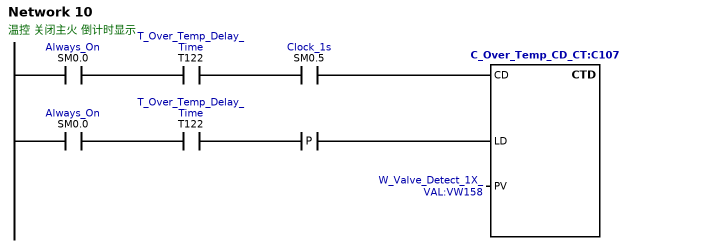
[picture p24: SBR4 networks 10-10]
Network 10
// 温控 关闭主火 倒计时显示
LD     Always_On:SM0.0
A      T_Over_Temp_Delay_Time:T122
A      Clock_1s:SM0.5
LD     Always_On:SM0.0
A      T_Over_Temp_Delay_Time:T122
EU
CTD    C_Over_Temp_CD_CT:C107, W_Valve_Detect_1X_VAL:VW158
END_SUBROUTINE_BLOCK

SUBROUTINE_BLOCK 阶段升温:SBR5
TITLE=
BEGIN
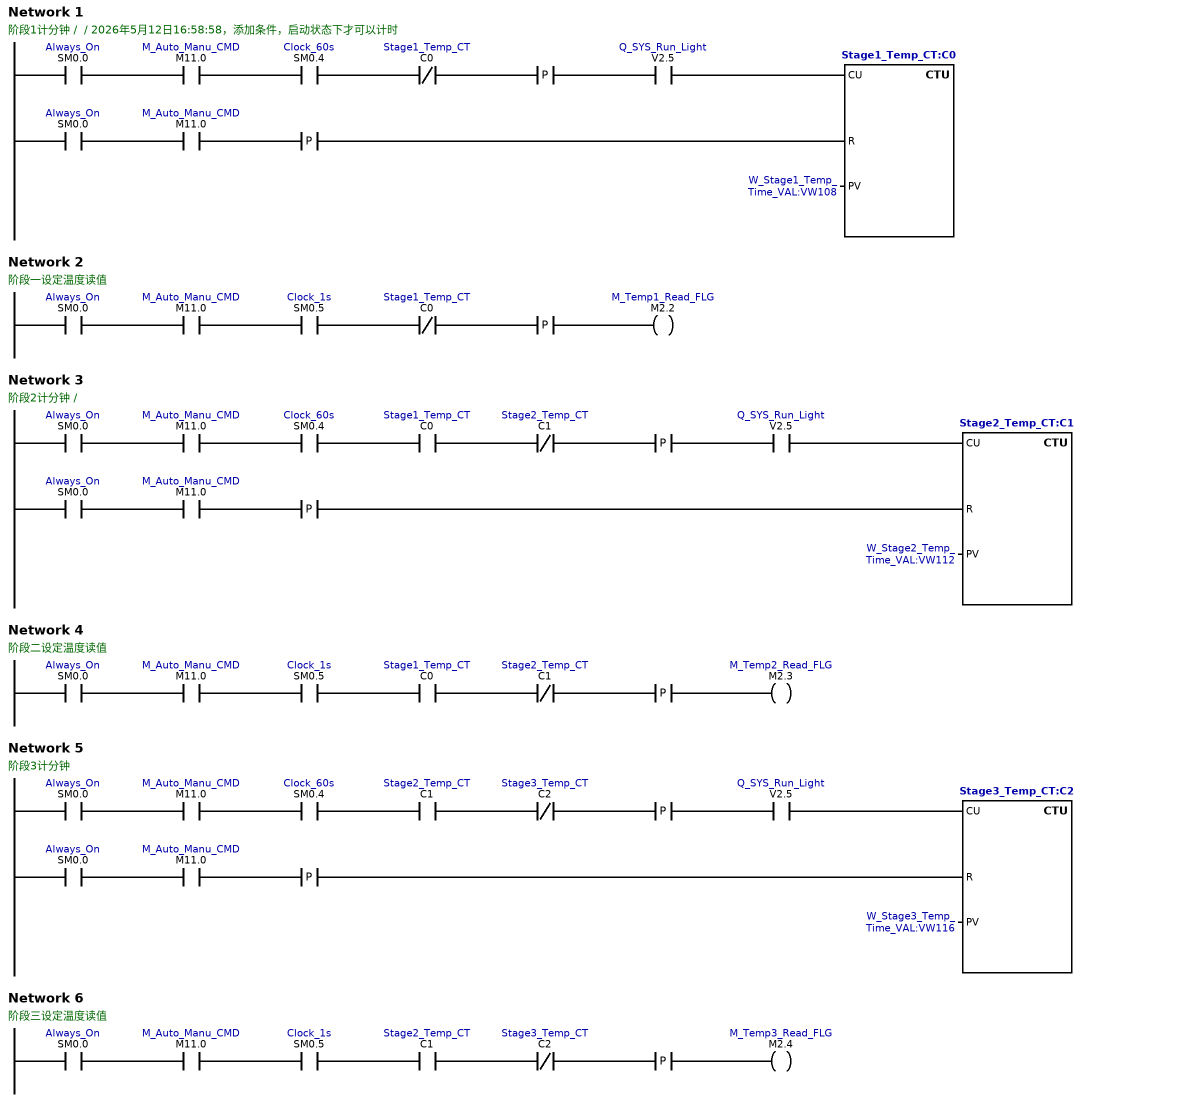
Network 1
// 阶段1计分钟
// 
// 2026年5月12日16:58:58，添加条件，启动状态下才可以计时
LD     Always_On:SM0.0
A      M_Auto_Manu_CMD:M11.0
A      Clock_60s:SM0.4
AN     Stage1_Temp_CT:C0
EU
A      Q_SYS_Run_Light:V2.5
LD     Always_On:SM0.0
A      M_Auto_Manu_CMD:M11.0
EU
CTU    Stage1_Temp_CT:C0, W_Stage1_Temp_Time_VAL:VW108
Network 2
// 阶段一设定温度读值
LD     Always_On:SM0.0
A      M_Auto_Manu_CMD:M11.0
A      Clock_1s:SM0.5
AN     Stage1_Temp_CT:C0
EU
=      M_Temp1_Read_FLG:M2.2
Network 3
// 阶段2计分钟
// 
LD     Always_On:SM0.0
A      M_Auto_Manu_CMD:M11.0
A      Clock_60s:SM0.4
A      Stage1_Temp_CT:C0
AN     Stage2_Temp_CT:C1
EU
A      Q_SYS_Run_Light:V2.5
LD     Always_On:SM0.0
A      M_Auto_Manu_CMD:M11.0
EU
CTU    Stage2_Temp_CT:C1, W_Stage2_Temp_Time_VAL:VW112
Network 4
// 阶段二设定温度读值
LD     Always_On:SM0.0
A      M_Auto_Manu_CMD:M11.0
A      Clock_1s:SM0.5
A      Stage1_Temp_CT:C0
AN     Stage2_Temp_CT:C1
EU
=      M_Temp2_Read_FLG:M2.3
Network 5
// 阶段3计分钟
LD     Always_On:SM0.0
A      M_Auto_Manu_CMD:M11.0
A      Clock_60s:SM0.4
A      Stage2_Temp_CT:C1
AN     Stage3_Temp_CT:C2
EU
A      Q_SYS_Run_Light:V2.5
LD     Always_On:SM0.0
A      M_Auto_Manu_CMD:M11.0
EU
CTU    Stage3_Temp_CT:C2, W_Stage3_Temp_Time_VAL:VW116
Network 6
// 阶段三设定温度读值
LD     Always_On:SM0.0
A      M_Auto_Manu_CMD:M11.0
A      Clock_1s:SM0.5
A      Stage2_Temp_CT:C1
AN     Stage3_Temp_CT:C2
EU
=      M_Temp3_Read_FLG:M2.4
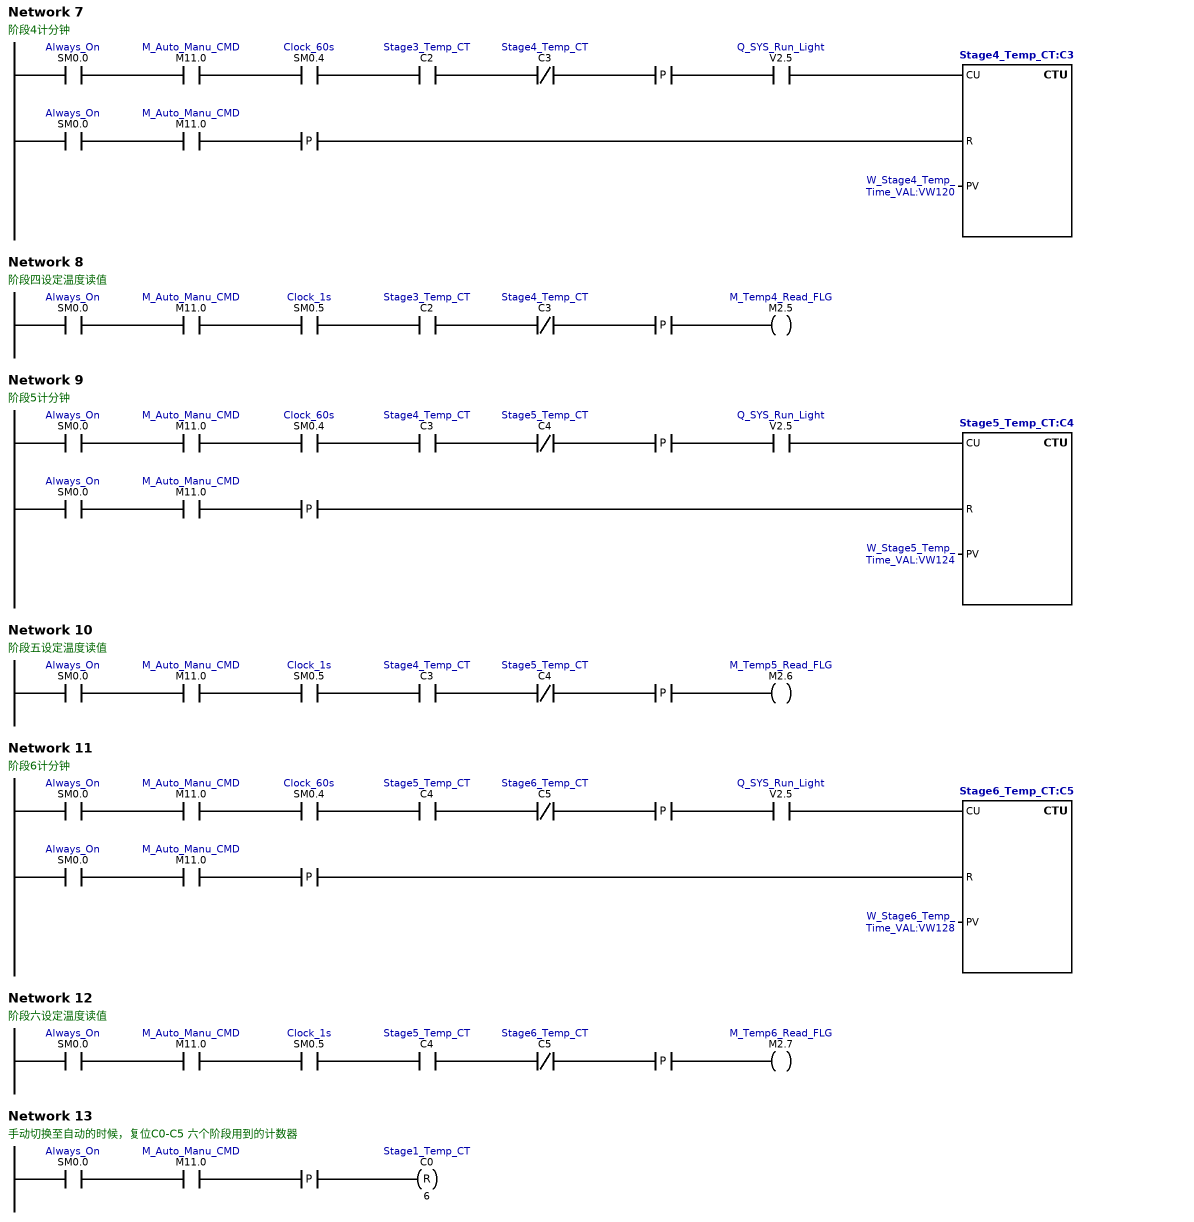
Network 7
// 阶段4计分钟
LD     Always_On:SM0.0
A      M_Auto_Manu_CMD:M11.0
A      Clock_60s:SM0.4
A      Stage3_Temp_CT:C2
AN     Stage4_Temp_CT:C3
EU
A      Q_SYS_Run_Light:V2.5
LD     Always_On:SM0.0
A      M_Auto_Manu_CMD:M11.0
EU
CTU    Stage4_Temp_CT:C3, W_Stage4_Temp_Time_VAL:VW120
Network 8
// 阶段四设定温度读值
LD     Always_On:SM0.0
A      M_Auto_Manu_CMD:M11.0
A      Clock_1s:SM0.5
A      Stage3_Temp_CT:C2
AN     Stage4_Temp_CT:C3
EU
=      M_Temp4_Read_FLG:M2.5
Network 9
// 阶段5计分钟
LD     Always_On:SM0.0
A      M_Auto_Manu_CMD:M11.0
A      Clock_60s:SM0.4
A      Stage4_Temp_CT:C3
AN     Stage5_Temp_CT:C4
EU
A      Q_SYS_Run_Light:V2.5
LD     Always_On:SM0.0
A      M_Auto_Manu_CMD:M11.0
EU
CTU    Stage5_Temp_CT:C4, W_Stage5_Temp_Time_VAL:VW124
Network 10
// 阶段五设定温度读值
LD     Always_On:SM0.0
A      M_Auto_Manu_CMD:M11.0
A      Clock_1s:SM0.5
A      Stage4_Temp_CT:C3
AN     Stage5_Temp_CT:C4
EU
=      M_Temp5_Read_FLG:M2.6
Network 11
// 阶段6计分钟
LD     Always_On:SM0.0
A      M_Auto_Manu_CMD:M11.0
A      Clock_60s:SM0.4
A      Stage5_Temp_CT:C4
AN     Stage6_Temp_CT:C5
EU
A      Q_SYS_Run_Light:V2.5
LD     Always_On:SM0.0
A      M_Auto_Manu_CMD:M11.0
EU
CTU    Stage6_Temp_CT:C5, W_Stage6_Temp_Time_VAL:VW128
Network 12
// 阶段六设定温度读值
LD     Always_On:SM0.0
A      M_Auto_Manu_CMD:M11.0
A      Clock_1s:SM0.5
A      Stage5_Temp_CT:C4
AN     Stage6_Temp_CT:C5
EU
=      M_Temp6_Read_FLG:M2.7
Network 13
// 手动切换至自动的时候，复位C0-C5 六个阶段用到的计数器
LD     Always_On:SM0.0
A      M_Auto_Manu_CMD:M11.0
EU
R      Stage1_Temp_CT:C0, 6
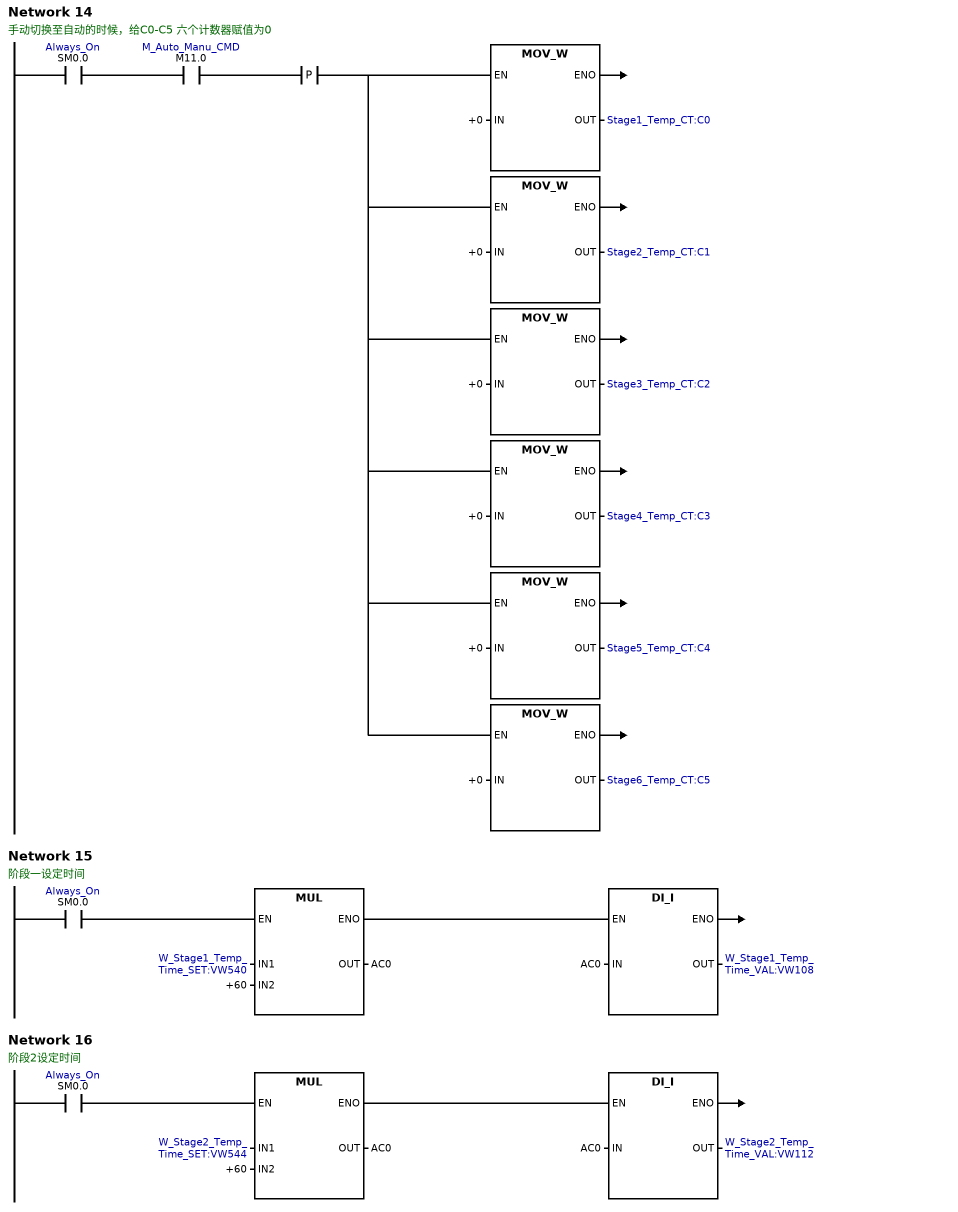
Network 14
// 手动切换至自动的时候，给C0-C5 六个计数器赋值为0
LD     Always_On:SM0.0
A      M_Auto_Manu_CMD:M11.0
EU
MOVW   +0, Stage1_Temp_CT:C0
MOVW   +0, Stage2_Temp_CT:C1
MOVW   +0, Stage3_Temp_CT:C2
MOVW   +0, Stage4_Temp_CT:C3
MOVW   +0, Stage5_Temp_CT:C4
MOVW   +0, Stage6_Temp_CT:C5
Network 15
// 阶段一设定时间
LD     Always_On:SM0.0
MOVW   W_Stage1_Temp_Time_SET:VW540, AC0
AENO
MUL    +60, AC0
AENO
DTI    AC0, W_Stage1_Temp_Time_VAL:VW108
Network 16
// 阶段2设定时间
LD     Always_On:SM0.0
MOVW   W_Stage2_Temp_Time_SET:VW544, AC0
AENO
MUL    +60, AC0
AENO
DTI    AC0, W_Stage2_Temp_Time_VAL:VW112
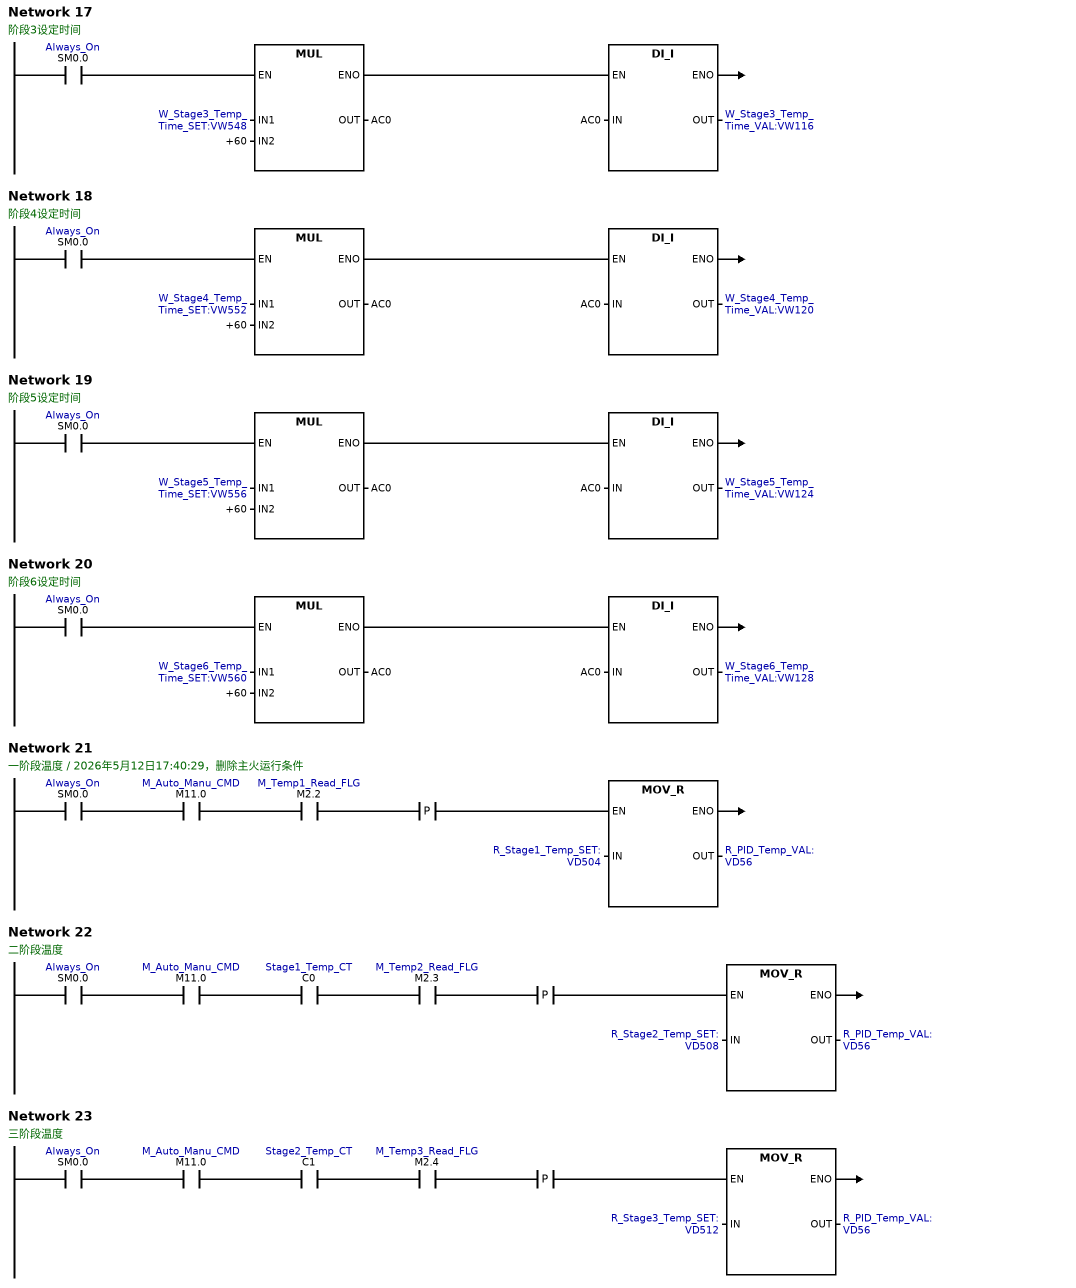
Network 17
// 阶段3设定时间
LD     Always_On:SM0.0
MOVW   W_Stage3_Temp_Time_SET:VW548, AC0
AENO
MUL    +60, AC0
AENO
DTI    AC0, W_Stage3_Temp_Time_VAL:VW116
Network 18
// 阶段4设定时间
LD     Always_On:SM0.0
MOVW   W_Stage4_Temp_Time_SET:VW552, AC0
AENO
MUL    +60, AC0
AENO
DTI    AC0, W_Stage4_Temp_Time_VAL:VW120
Network 19
// 阶段5设定时间
LD     Always_On:SM0.0
MOVW   W_Stage5_Temp_Time_SET:VW556, AC0
AENO
MUL    +60, AC0
AENO
DTI    AC0, W_Stage5_Temp_Time_VAL:VW124
Network 20
// 阶段6设定时间
LD     Always_On:SM0.0
MOVW   W_Stage6_Temp_Time_SET:VW560, AC0
AENO
MUL    +60, AC0
AENO
DTI    AC0, W_Stage6_Temp_Time_VAL:VW128
Network 21
// 一阶段温度
// 2026年5月12日17:40:29，删除主火运行条件
LD     Always_On:SM0.0
A      M_Auto_Manu_CMD:M11.0
A      M_Temp1_Read_FLG:M2.2
EU
MOVR   R_Stage1_Temp_SET:VD504, R_PID_Temp_VAL:VD56
Network 22
// 二阶段温度
LD     Always_On:SM0.0
A      M_Auto_Manu_CMD:M11.0
A      Stage1_Temp_CT:C0
A      M_Temp2_Read_FLG:M2.3
EU
MOVR   R_Stage2_Temp_SET:VD508, R_PID_Temp_VAL:VD56
Network 23
// 三阶段温度
LD     Always_On:SM0.0
A      M_Auto_Manu_CMD:M11.0
A      Stage2_Temp_CT:C1
A      M_Temp3_Read_FLG:M2.4
EU
MOVR   R_Stage3_Temp_SET:VD512, R_PID_Temp_VAL:VD56
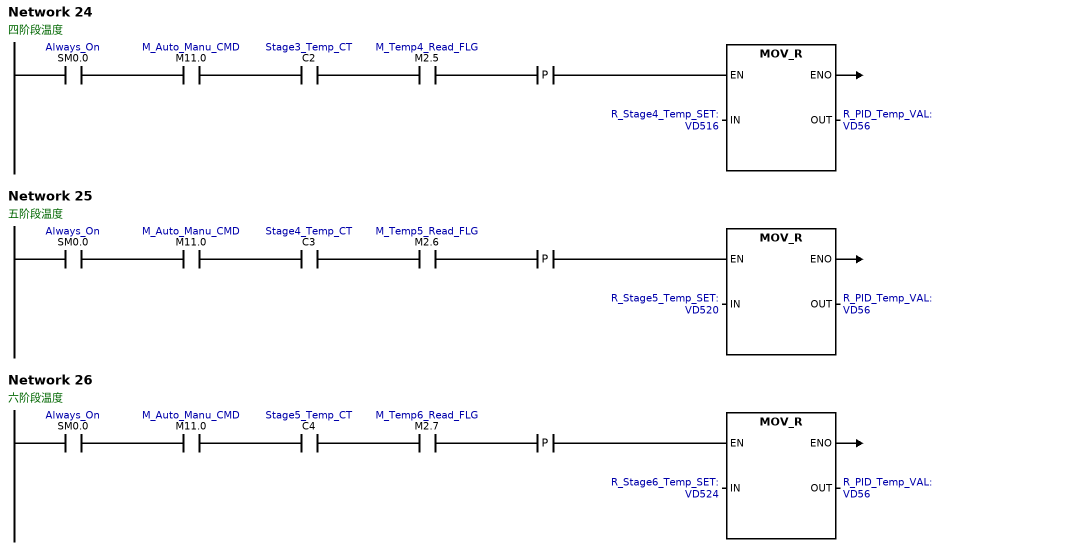
Network 24
// 四阶段温度
LD     Always_On:SM0.0
A      M_Auto_Manu_CMD:M11.0
A      Stage3_Temp_CT:C2
A      M_Temp4_Read_FLG:M2.5
EU
MOVR   R_Stage4_Temp_SET:VD516, R_PID_Temp_VAL:VD56
Network 25
// 五阶段温度
LD     Always_On:SM0.0
A      M_Auto_Manu_CMD:M11.0
A      Stage4_Temp_CT:C3
A      M_Temp5_Read_FLG:M2.6
EU
MOVR   R_Stage5_Temp_SET:VD520, R_PID_Temp_VAL:VD56
Network 26
// 六阶段温度
LD     Always_On:SM0.0
A      M_Auto_Manu_CMD:M11.0
A      Stage5_Temp_CT:C4
A      M_Temp6_Read_FLG:M2.7
EU
MOVR   R_Stage6_Temp_SET:VD524, R_PID_Temp_VAL:VD56
END_SUBROUTINE_BLOCK

SUBROUTINE_BLOCK 开度档位:SBR6
TITLE=开度档位子程序
// 功能：
// 1、处理每档对应的燃气调节阀开度多少，空气调节阀开度多少。
// 2、手动模式，升档、降档控制
// 3、自动模式，PID输出转换成档位处理
// 
BEGIN
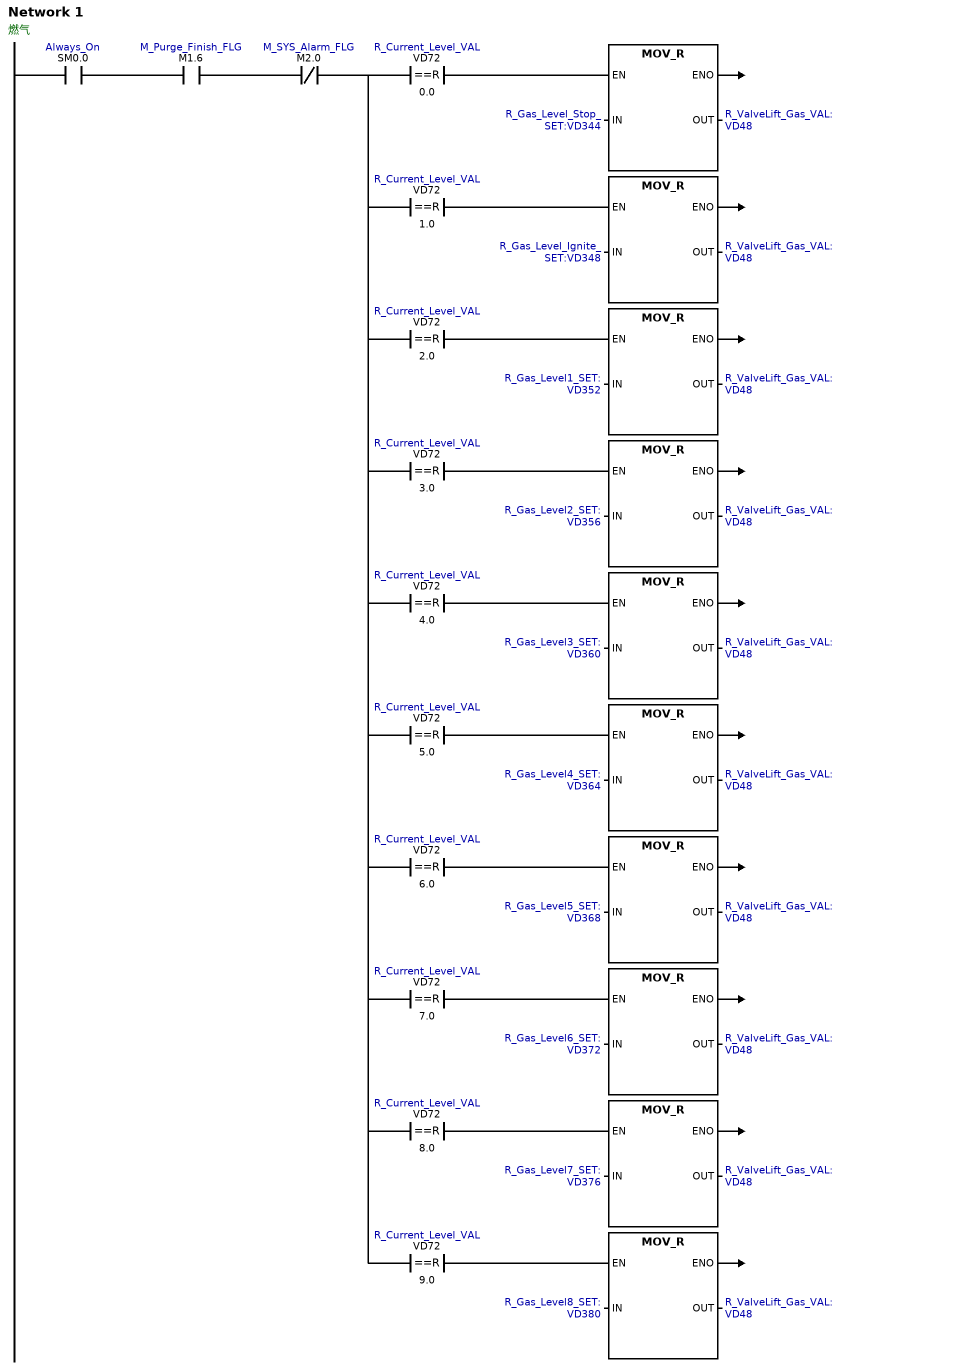
Network 1
// 燃气
LD     Always_On:SM0.0
A      M_Purge_Finish_FLG:M1.6
AN     M_SYS_Alarm_FLG:M2.0
LPS
AR=    R_Current_Level_VAL:VD72, 0.0
MOVR   R_Gas_Level_Stop_SET:VD344, R_ValveLift_Gas_VAL:VD48
LRD
AR=    R_Current_Level_VAL:VD72, 1.0
MOVR   R_Gas_Level_Ignite_SET:VD348, R_ValveLift_Gas_VAL:VD48
LRD
AR=    R_Current_Level_VAL:VD72, 2.0
MOVR   R_Gas_Level1_SET:VD352, R_ValveLift_Gas_VAL:VD48
LRD
AR=    R_Current_Level_VAL:VD72, 3.0
MOVR   R_Gas_Level2_SET:VD356, R_ValveLift_Gas_VAL:VD48
LRD
AR=    R_Current_Level_VAL:VD72, 4.0
MOVR   R_Gas_Level3_SET:VD360, R_ValveLift_Gas_VAL:VD48
LRD
AR=    R_Current_Level_VAL:VD72, 5.0
MOVR   R_Gas_Level4_SET:VD364, R_ValveLift_Gas_VAL:VD48
LRD
AR=    R_Current_Level_VAL:VD72, 6.0
MOVR   R_Gas_Level5_SET:VD368, R_ValveLift_Gas_VAL:VD48
LRD
AR=    R_Current_Level_VAL:VD72, 7.0
MOVR   R_Gas_Level6_SET:VD372, R_ValveLift_Gas_VAL:VD48
LRD
AR=    R_Current_Level_VAL:VD72, 8.0
MOVR   R_Gas_Level7_SET:VD376, R_ValveLift_Gas_VAL:VD48
LPP
AR=    R_Current_Level_VAL:VD72, 9.0
MOVR   R_Gas_Level8_SET:VD380, R_ValveLift_Gas_VAL:VD48
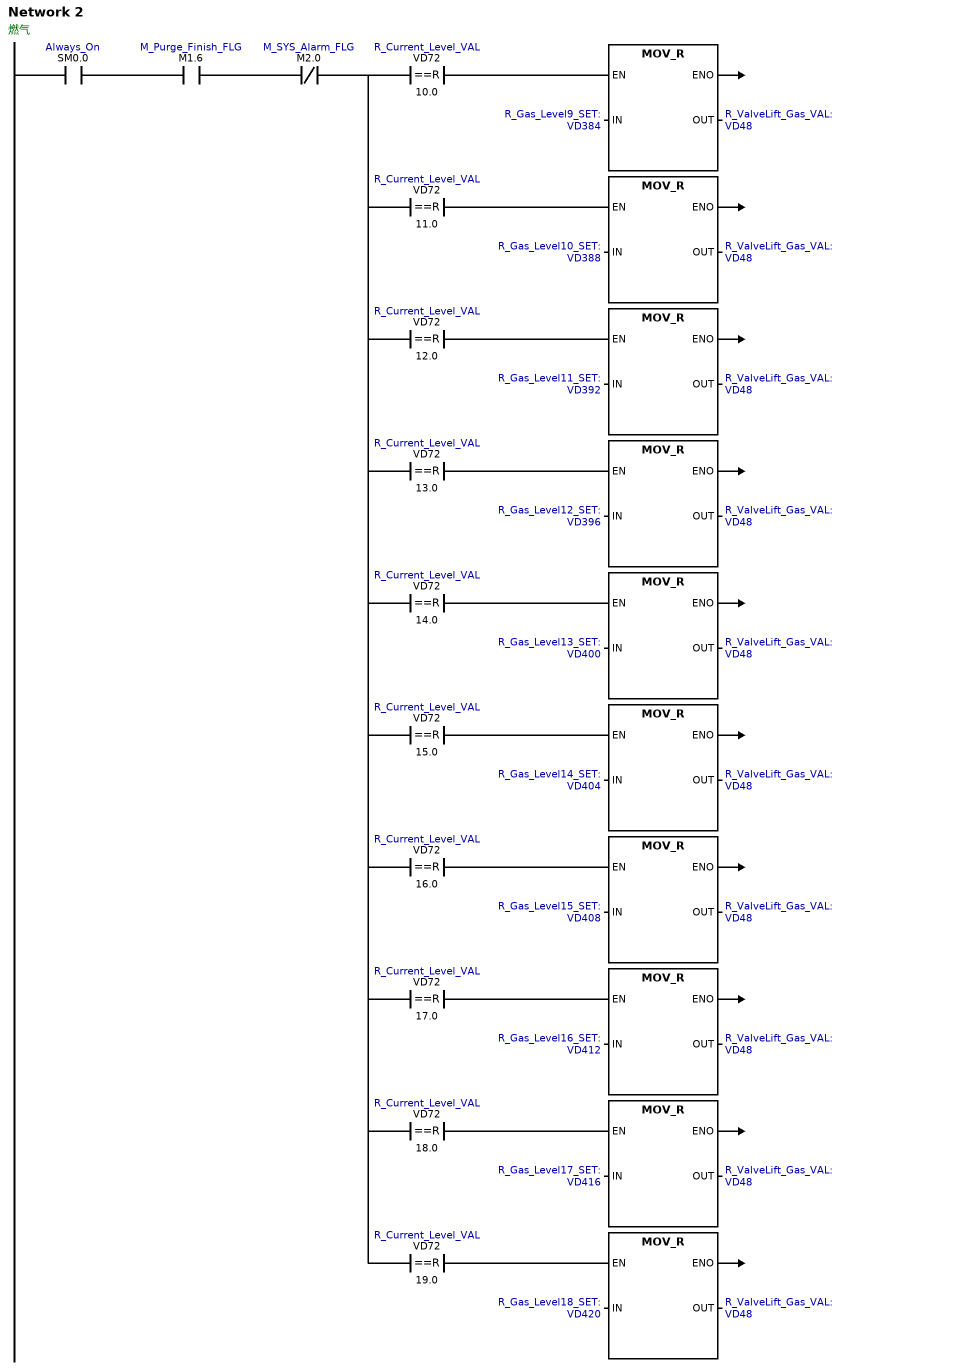
Network 2
// 燃气
LD     Always_On:SM0.0
A      M_Purge_Finish_FLG:M1.6
AN     M_SYS_Alarm_FLG:M2.0
LPS
AR=    R_Current_Level_VAL:VD72, 10.0
MOVR   R_Gas_Level9_SET:VD384, R_ValveLift_Gas_VAL:VD48
LRD
AR=    R_Current_Level_VAL:VD72, 11.0
MOVR   R_Gas_Level10_SET:VD388, R_ValveLift_Gas_VAL:VD48
LRD
AR=    R_Current_Level_VAL:VD72, 12.0
MOVR   R_Gas_Level11_SET:VD392, R_ValveLift_Gas_VAL:VD48
LRD
AR=    R_Current_Level_VAL:VD72, 13.0
MOVR   R_Gas_Level12_SET:VD396, R_ValveLift_Gas_VAL:VD48
LRD
AR=    R_Current_Level_VAL:VD72, 14.0
MOVR   R_Gas_Level13_SET:VD400, R_ValveLift_Gas_VAL:VD48
LRD
AR=    R_Current_Level_VAL:VD72, 15.0
MOVR   R_Gas_Level14_SET:VD404, R_ValveLift_Gas_VAL:VD48
LRD
AR=    R_Current_Level_VAL:VD72, 16.0
MOVR   R_Gas_Level15_SET:VD408, R_ValveLift_Gas_VAL:VD48
LRD
AR=    R_Current_Level_VAL:VD72, 17.0
MOVR   R_Gas_Level16_SET:VD412, R_ValveLift_Gas_VAL:VD48
LRD
AR=    R_Current_Level_VAL:VD72, 18.0
MOVR   R_Gas_Level17_SET:VD416, R_ValveLift_Gas_VAL:VD48
LPP
AR=    R_Current_Level_VAL:VD72, 19.0
MOVR   R_Gas_Level18_SET:VD420, R_ValveLift_Gas_VAL:VD48
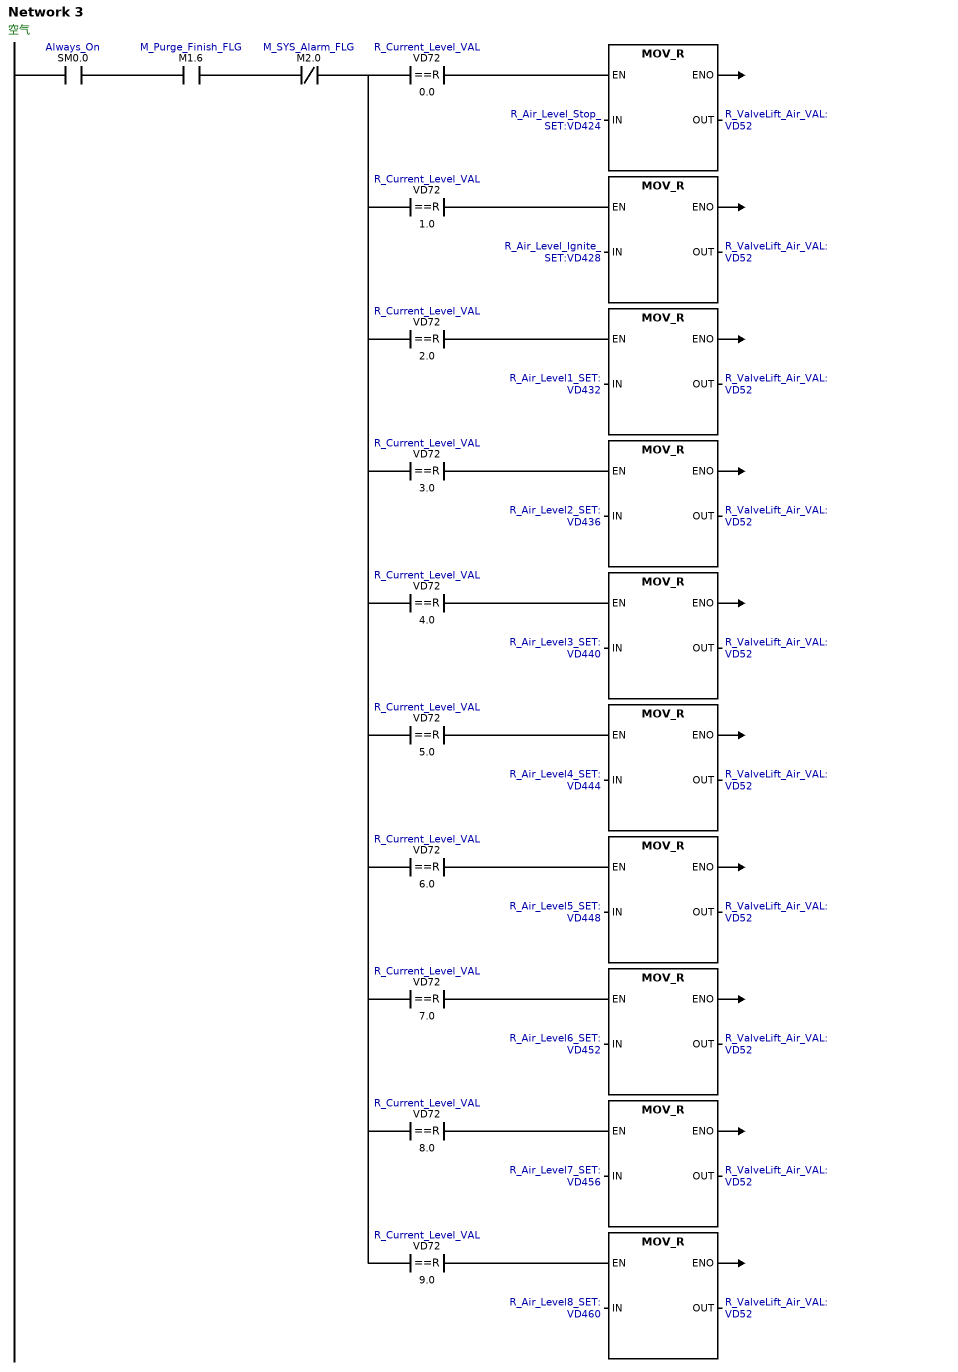
Network 3
// 空气
LD     Always_On:SM0.0
A      M_Purge_Finish_FLG:M1.6
AN     M_SYS_Alarm_FLG:M2.0
LPS
AR=    R_Current_Level_VAL:VD72, 0.0
MOVR   R_Air_Level_Stop_SET:VD424, R_ValveLift_Air_VAL:VD52
LRD
AR=    R_Current_Level_VAL:VD72, 1.0
MOVR   R_Air_Level_Ignite_SET:VD428, R_ValveLift_Air_VAL:VD52
LRD
AR=    R_Current_Level_VAL:VD72, 2.0
MOVR   R_Air_Level1_SET:VD432, R_ValveLift_Air_VAL:VD52
LRD
AR=    R_Current_Level_VAL:VD72, 3.0
MOVR   R_Air_Level2_SET:VD436, R_ValveLift_Air_VAL:VD52
LRD
AR=    R_Current_Level_VAL:VD72, 4.0
MOVR   R_Air_Level3_SET:VD440, R_ValveLift_Air_VAL:VD52
LRD
AR=    R_Current_Level_VAL:VD72, 5.0
MOVR   R_Air_Level4_SET:VD444, R_ValveLift_Air_VAL:VD52
LRD
AR=    R_Current_Level_VAL:VD72, 6.0
MOVR   R_Air_Level5_SET:VD448, R_ValveLift_Air_VAL:VD52
LRD
AR=    R_Current_Level_VAL:VD72, 7.0
MOVR   R_Air_Level6_SET:VD452, R_ValveLift_Air_VAL:VD52
LRD
AR=    R_Current_Level_VAL:VD72, 8.0
MOVR   R_Air_Level7_SET:VD456, R_ValveLift_Air_VAL:VD52
LPP
AR=    R_Current_Level_VAL:VD72, 9.0
MOVR   R_Air_Level8_SET:VD460, R_ValveLift_Air_VAL:VD52
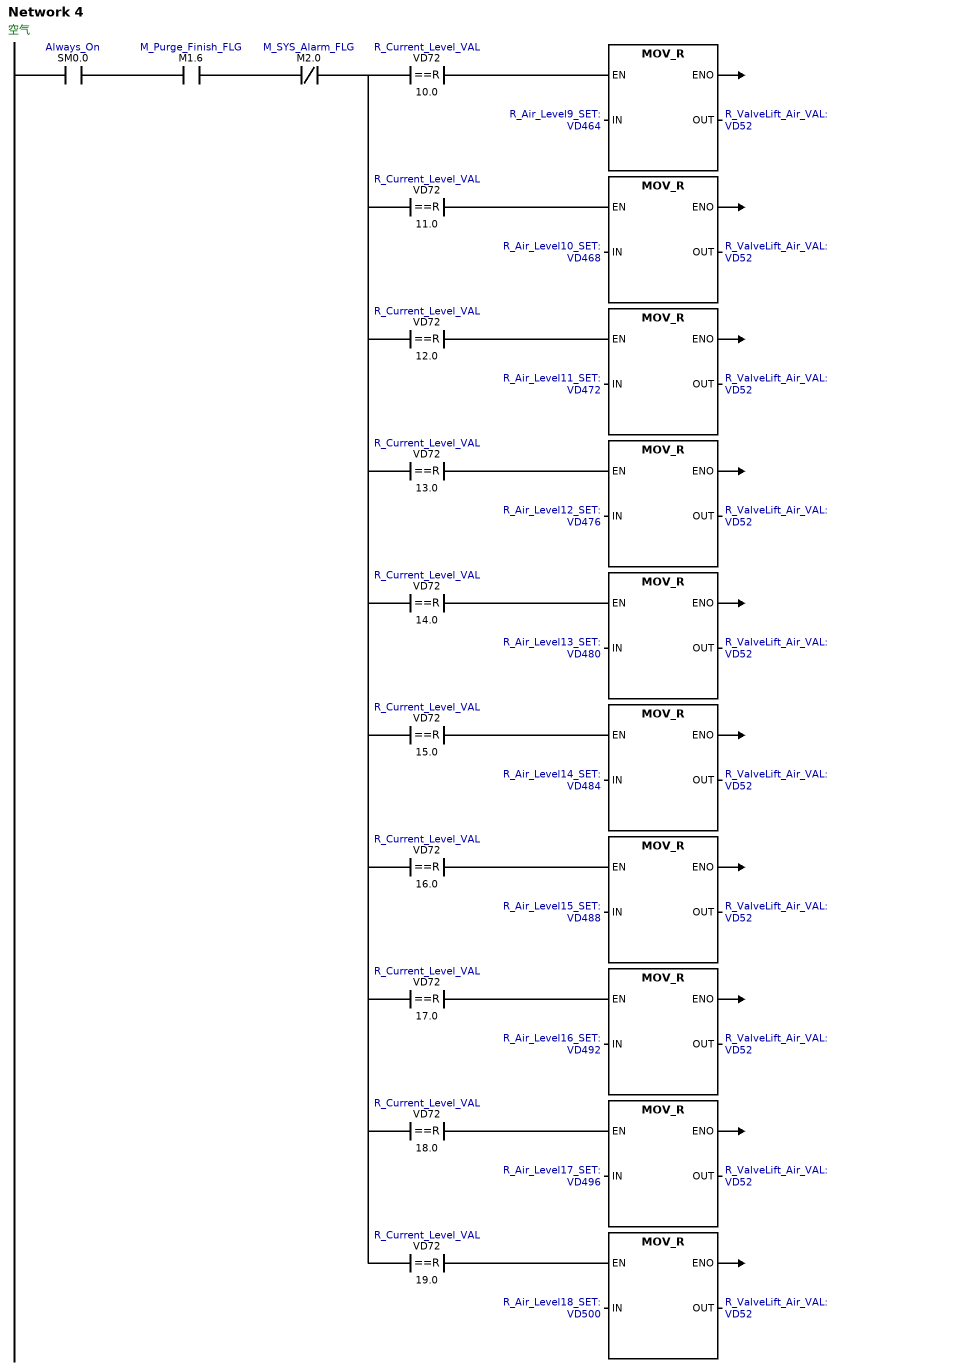
Network 4
// 空气
LD     Always_On:SM0.0
A      M_Purge_Finish_FLG:M1.6
AN     M_SYS_Alarm_FLG:M2.0
LPS
AR=    R_Current_Level_VAL:VD72, 10.0
MOVR   R_Air_Level9_SET:VD464, R_ValveLift_Air_VAL:VD52
LRD
AR=    R_Current_Level_VAL:VD72, 11.0
MOVR   R_Air_Level10_SET:VD468, R_ValveLift_Air_VAL:VD52
LRD
AR=    R_Current_Level_VAL:VD72, 12.0
MOVR   R_Air_Level11_SET:VD472, R_ValveLift_Air_VAL:VD52
LRD
AR=    R_Current_Level_VAL:VD72, 13.0
MOVR   R_Air_Level12_SET:VD476, R_ValveLift_Air_VAL:VD52
LRD
AR=    R_Current_Level_VAL:VD72, 14.0
MOVR   R_Air_Level13_SET:VD480, R_ValveLift_Air_VAL:VD52
LRD
AR=    R_Current_Level_VAL:VD72, 15.0
MOVR   R_Air_Level14_SET:VD484, R_ValveLift_Air_VAL:VD52
LRD
AR=    R_Current_Level_VAL:VD72, 16.0
MOVR   R_Air_Level15_SET:VD488, R_ValveLift_Air_VAL:VD52
LRD
AR=    R_Current_Level_VAL:VD72, 17.0
MOVR   R_Air_Level16_SET:VD492, R_ValveLift_Air_VAL:VD52
LRD
AR=    R_Current_Level_VAL:VD72, 18.0
MOVR   R_Air_Level17_SET:VD496, R_ValveLift_Air_VAL:VD52
LPP
AR=    R_Current_Level_VAL:VD72, 19.0
MOVR   R_Air_Level18_SET:VD500, R_ValveLift_Air_VAL:VD52
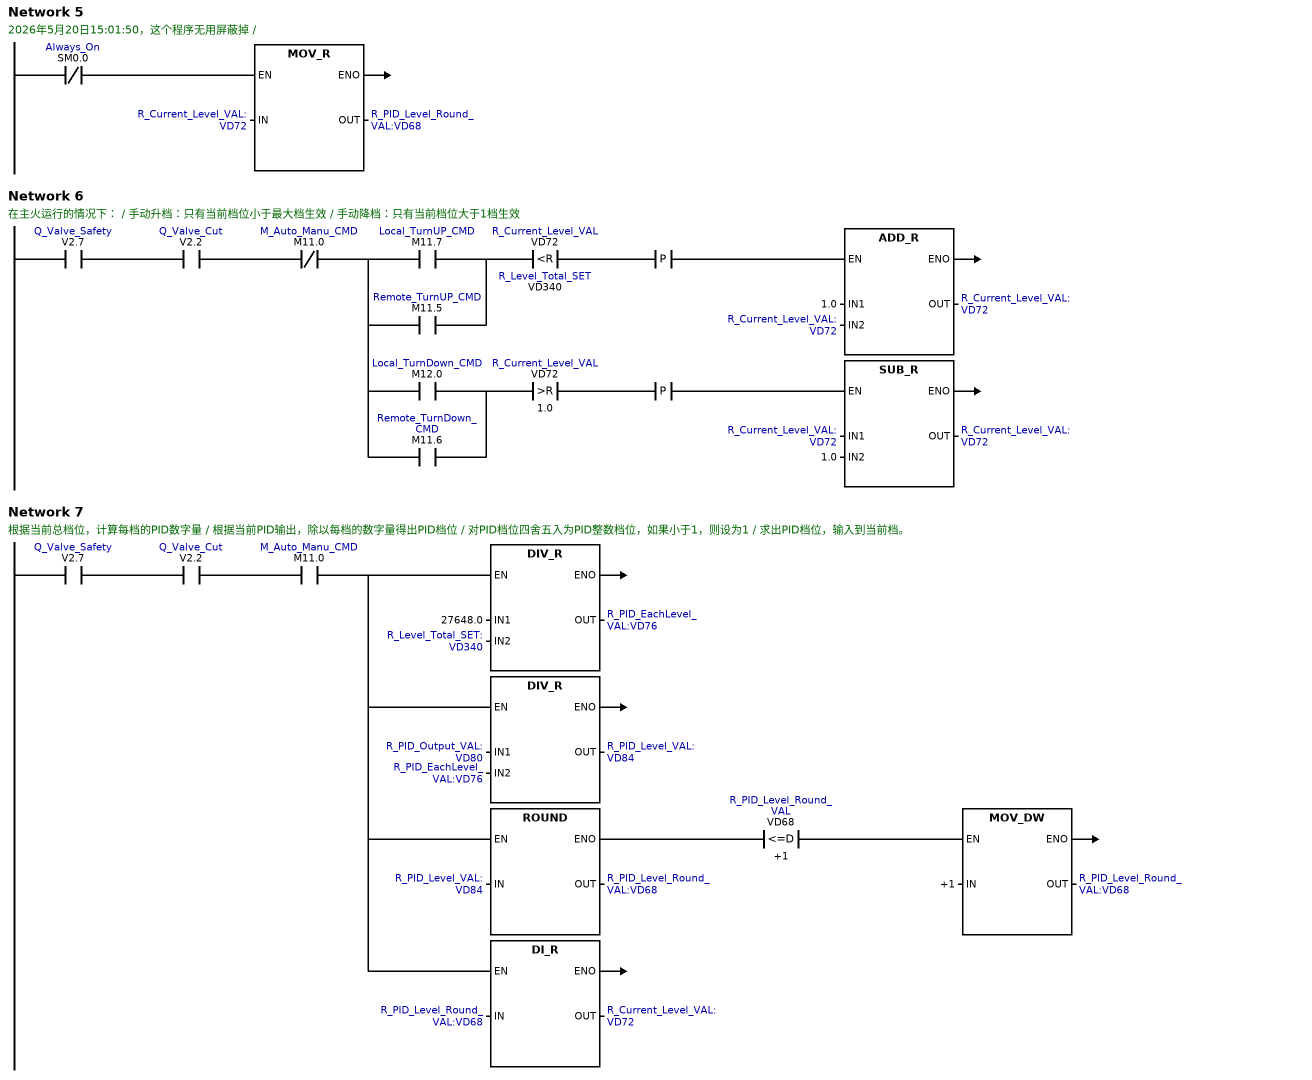
Network 5
// 2026年5月20日15:01:50，这个程序无用屏蔽掉
// 
LDN    Always_On:SM0.0
MOVR   R_Current_Level_VAL:VD72, R_PID_Level_Round_VAL:VD68
Network 6
// 在主火运行的情况下：
// 手动升档：只有当前档位小于最大档生效
// 手动降档：只有当前档位大于1档生效
LD     Q_Valve_Safety:V2.7
A      Q_Valve_Cut:V2.2
AN     M_Auto_Manu_CMD:M11.0
LPS
LD     Local_TurnUP_CMD:M11.7
O      Remote_TurnUP_CMD:M11.5
ALD
AR<    R_Current_Level_VAL:VD72, R_Level_Total_SET:VD340
EU
+R     1.0, R_Current_Level_VAL:VD72
LPP
LD     Local_TurnDown_CMD:M12.0
O      Remote_TurnDown_CMD:M11.6
ALD
AR>    R_Current_Level_VAL:VD72, 1.0
EU
-R     1.0, R_Current_Level_VAL:VD72
Network 7
// 根据当前总档位，计算每档的PID数字量
// 根据当前PID输出，除以每档的数字量得出PID档位
// 对PID档位四舍五入为PID整数档位，如果小于1，则设为1
// 求出PID档位，输入到当前档。
LD     Q_Valve_Safety:V2.7
A      Q_Valve_Cut:V2.2
A      M_Auto_Manu_CMD:M11.0
LPS
MOVR   27648.0, R_PID_EachLevel_VAL:VD76
/R     R_Level_Total_SET:VD340, R_PID_EachLevel_VAL:VD76
MOVR   R_PID_Output_VAL:VD80, R_PID_Level_VAL:VD84
/R     R_PID_EachLevel_VAL:VD76, R_PID_Level_VAL:VD84
ROUND  R_PID_Level_VAL:VD84, R_PID_Level_Round_VAL:VD68
AENO
AD<=   R_PID_Level_Round_VAL:VD68, +1
MOVD   +1, R_PID_Level_Round_VAL:VD68
LPP
DTR    R_PID_Level_Round_VAL:VD68, R_Current_Level_VAL:VD72
END_SUBROUTINE_BLOCK

SUBROUTINE_BLOCK 远程通讯:SBR7
TITLE=远程通讯子程序
// 功能：
// 1、初始化从站（PLC）
// 	模式Mode（通讯协议）：	1、Modubs协议；0、PPI协
// 	地址Addr	：	1-247
// 	波特率Baud：	1200、2400、4800、9600、19200、38400、57600、11500
// 	奇偶校验Parity：	0无校验、1奇校验、2偶校验
// 	端口Port：	0=CPU集成RS-485端口，1=可选信号板上的RS-485或RS-232
// 	延时Delay：	可以是0-32767
// 	MaxIQ：		设置Modbus地址0XXXX和1XXXX可用 的I和Q点数，0-256
// 	MaxAI：		设置Modbus地址3XXXX可用的字输入（AI）寄存器数，0（CR系列）或56（其它系列）
// 	MaxHold：	设置Modbus地址4XXXX或4yyyyy可访问的V存储器中的字保持寄存器数。如果要允许 Modbus 主站访问 2000 个字节的 V 存储器，请将 MaxHold的值设置为 1000 个字（保持寄存器）
// 	HoldStart：	是 V 存储器中保持寄存器的起始地址	
// 
// 2、处理主站请求
// 在每次扫描处理主站请求
// 
// 
// 
// 3、显示设备状态：
// 	故障状态RTU
// 	自动状态RTU
// 	启动状态RTU
// 	停止状态RTU
// 	本地远程状态RTU
// 
// 4、处理DCS传送过来的温度数据,VW1898
BEGIN
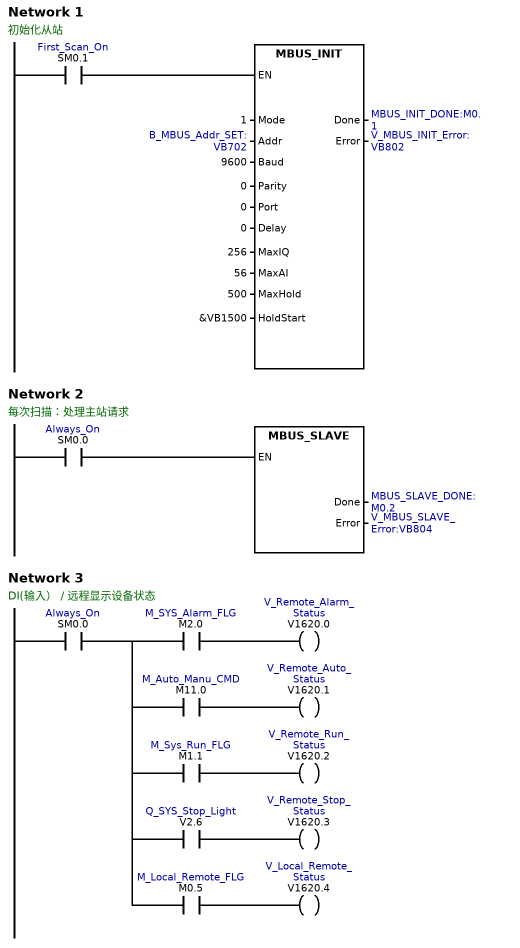
Network 1
// 初始化从站
LD     First_Scan_On:SM0.1
CALL   MBUS_INIT:SBR21, 1, B_MBUS_Addr_SET:VB702, 9600, 0, 0, 0, 256, 56, 500, &VB1500, MBUS_INIT_DONE:M0.1, V_MBUS_INIT_Error:VB802
Network 2
// 每次扫描：处理主站请求
LD     Always_On:SM0.0
CALL   MBUS_SLAVE:SBR22, MBUS_SLAVE_DONE:M0.2, V_MBUS_SLAVE_Error:VB804
Network 3
// DI(输入）
// 远程显示设备状态
LD     Always_On:SM0.0
LPS
A      M_SYS_Alarm_FLG:M2.0
=      V_Remote_Alarm_Status:V1620.0
LRD
A      M_Auto_Manu_CMD:M11.0
=      V_Remote_Auto_Status:V1620.1
LRD
A      M_Sys_Run_FLG:M1.1
=      V_Remote_Run_Status:V1620.2
LRD
A      Q_SYS_Stop_Light:V2.6
=      V_Remote_Stop_Status:V1620.3
LPP
A      M_Local_Remote_FLG:M0.5
=      V_Local_Remote_Status:V1620.4
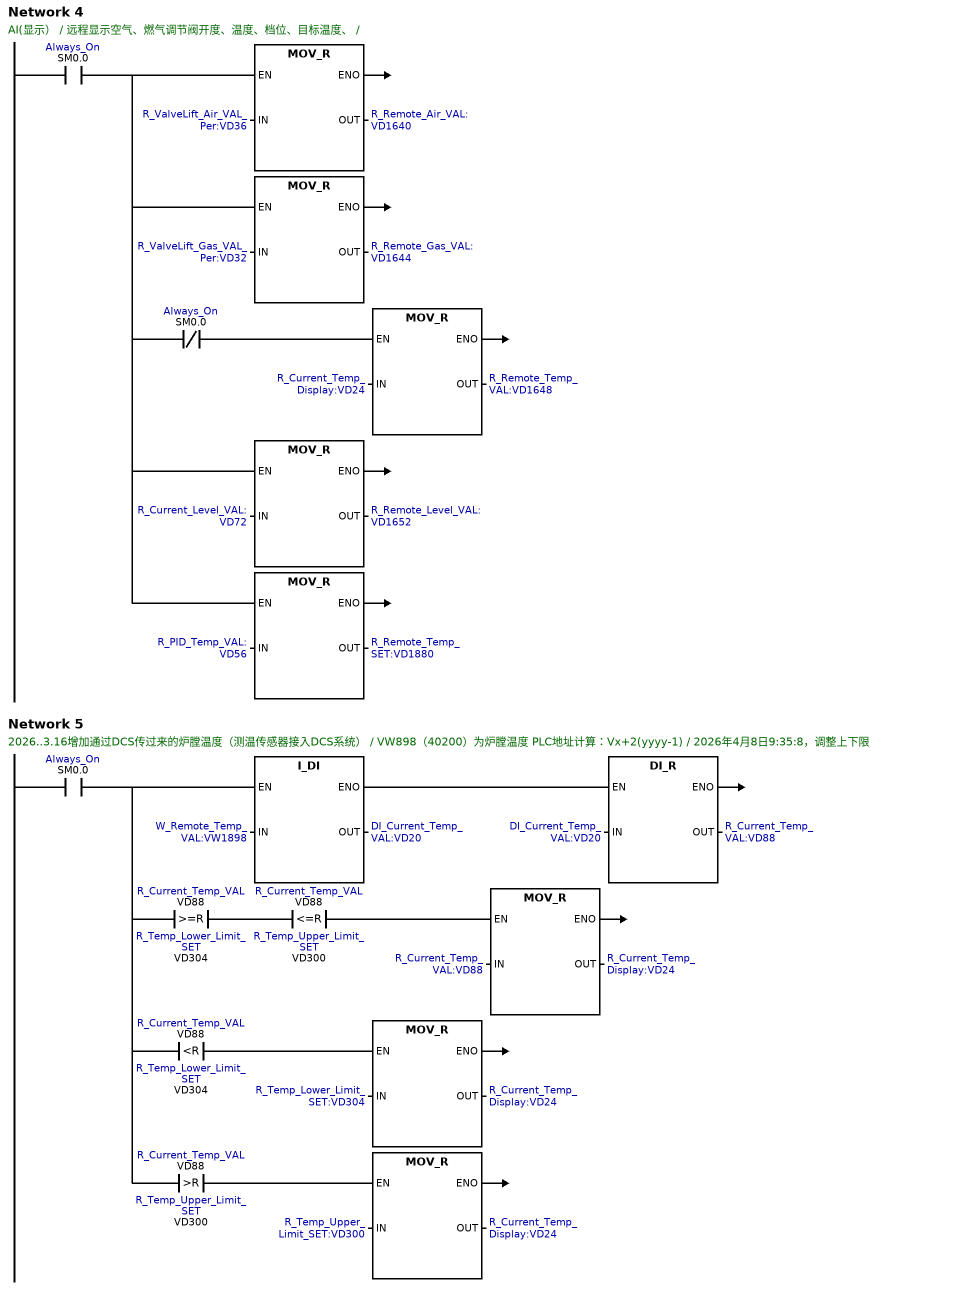
Network 4
// AI(显示）
// 远程显示空气、燃气调节阀开度、温度、档位、目标温度、
// 
LD     Always_On:SM0.0
LPS
MOVR   R_ValveLift_Air_VAL_Per:VD36, R_Remote_Air_VAL:VD1640
MOVR   R_ValveLift_Gas_VAL_Per:VD32, R_Remote_Gas_VAL:VD1644
AN     Always_On:SM0.0
MOVR   R_Current_Temp_Display:VD24, R_Remote_Temp_VAL:VD1648
LRD
MOVR   R_Current_Level_VAL:VD72, R_Remote_Level_VAL:VD1652
LPP
MOVR   R_PID_Temp_VAL:VD56, R_Remote_Temp_SET:VD1880
Network 5
// 2026..3.16增加通过DCS传过来的炉膛温度（测温传感器接入DCS系统）
// VW898（40200）为炉膛温度 PLC地址计算：Vx+2(yyyy-1)
// 2026年4月8日9:35:8，调整上下限
LD     Always_On:SM0.0
LPS
ITD    W_Remote_Temp_VAL:VW1898, DI_Current_Temp_VAL:VD20
AENO
DTR    DI_Current_Temp_VAL:VD20, R_Current_Temp_VAL:VD88
LRD
AR>=   R_Current_Temp_VAL:VD88, R_Temp_Lower_Limit_SET:VD304
AR<=   R_Current_Temp_VAL:VD88, R_Temp_Upper_Limit_SET:VD300
MOVR   R_Current_Temp_VAL:VD88, R_Current_Temp_Display:VD24
LRD
AR<    R_Current_Temp_VAL:VD88, R_Temp_Lower_Limit_SET:VD304
MOVR   R_Temp_Lower_Limit_SET:VD304, R_Current_Temp_Display:VD24
LPP
AR>    R_Current_Temp_VAL:VD88, R_Temp_Upper_Limit_SET:VD300
MOVR   R_Temp_Upper_Limit_SET:VD300, R_Current_Temp_Display:VD24
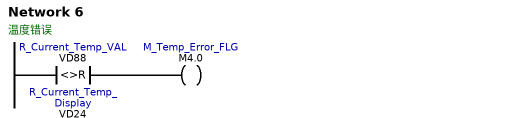
Network 6
// 温度错误
LDR<>  R_Current_Temp_VAL:VD88, R_Current_Temp_Display:VD24
=      M_Temp_Error_FLG:M4.0
END_SUBROUTINE_BLOCK

SUBROUTINE_BLOCK IO设备:SBR8
TITLE=子程序注释
// 1、IO映射
// 2、统一输出
// 	蜂鸣器
// 	点火阀
// 	主火阀V2
// 	点火变压器
// 	有火指示灯
// 	启动指示灯
// 	停止指示灯
// 	安全阀V1
// 
// 
BEGIN
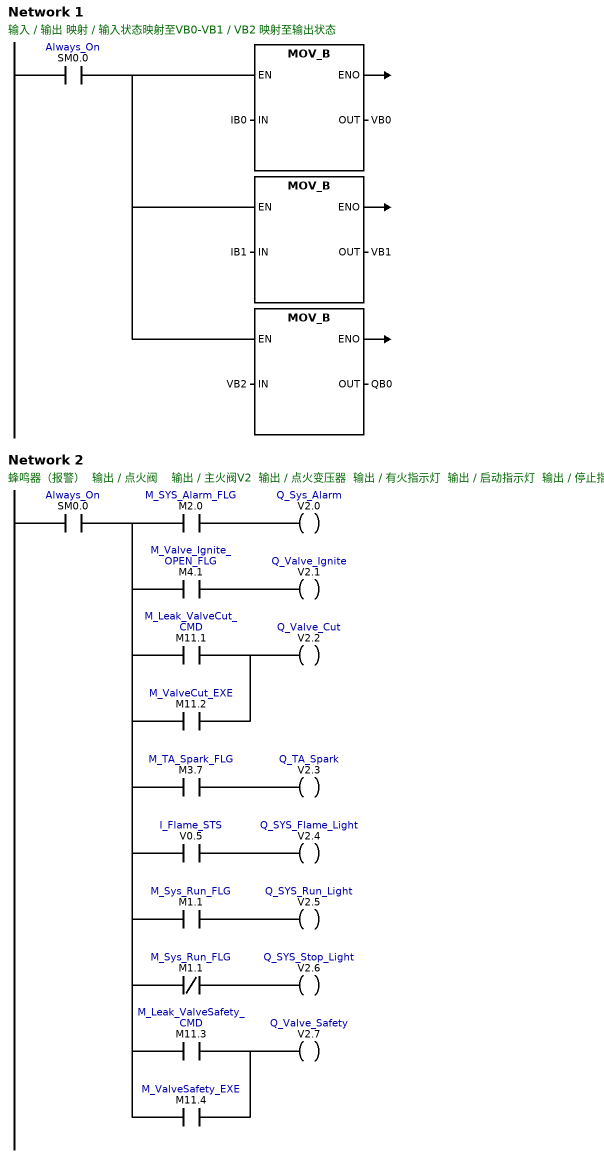
Network 1
// 输入 / 输出 映射
// 输入状态映射至VB0-VB1
// VB2 映射至输出状态
LD     Always_On:SM0.0
MOVB   IB0, VB0
MOVB   IB1, VB1
MOVB   VB2, QB0
Network 2
// 蜂鸣器（报警）	输出
// 点火阀		输出
// 主火阀V2	输出
// 点火变压器	输出
// 有火指示灯	输出
// 启动指示灯	输出
// 停止指示灯	输出
// 安全阀V1	输出
// 
LD     Always_On:SM0.0
LPS
A      M_SYS_Alarm_FLG:M2.0
=      Q_Sys_Alarm:V2.0
LRD
A      M_Valve_Ignite_OPEN_FLG:M4.1
=      Q_Valve_Ignite:V2.1
LRD
LD     M_Leak_ValveCut_CMD:M11.1
O      M_ValveCut_EXE:M11.2
ALD
=      Q_Valve_Cut:V2.2
LRD
LPS
A      M_TA_Spark_FLG:M3.7
=      Q_TA_Spark:V2.3
LRD
A      I_Flame_STS:V0.5
=      Q_SYS_Flame_Light:V2.4
LRD
A      M_Sys_Run_FLG:M1.1
=      Q_SYS_Run_Light:V2.5
LPP
AN     M_Sys_Run_FLG:M1.1
=      Q_SYS_Stop_Light:V2.6
LPP
LD     M_Leak_ValveSafety_CMD:M11.3
O      M_ValveSafety_EXE:M11.4
ALD
=      Q_Valve_Safety:V2.7
END_SUBROUTINE_BLOCK

SUBROUTINE_BLOCK 运行时间:SBR9
TITLE=
BEGIN
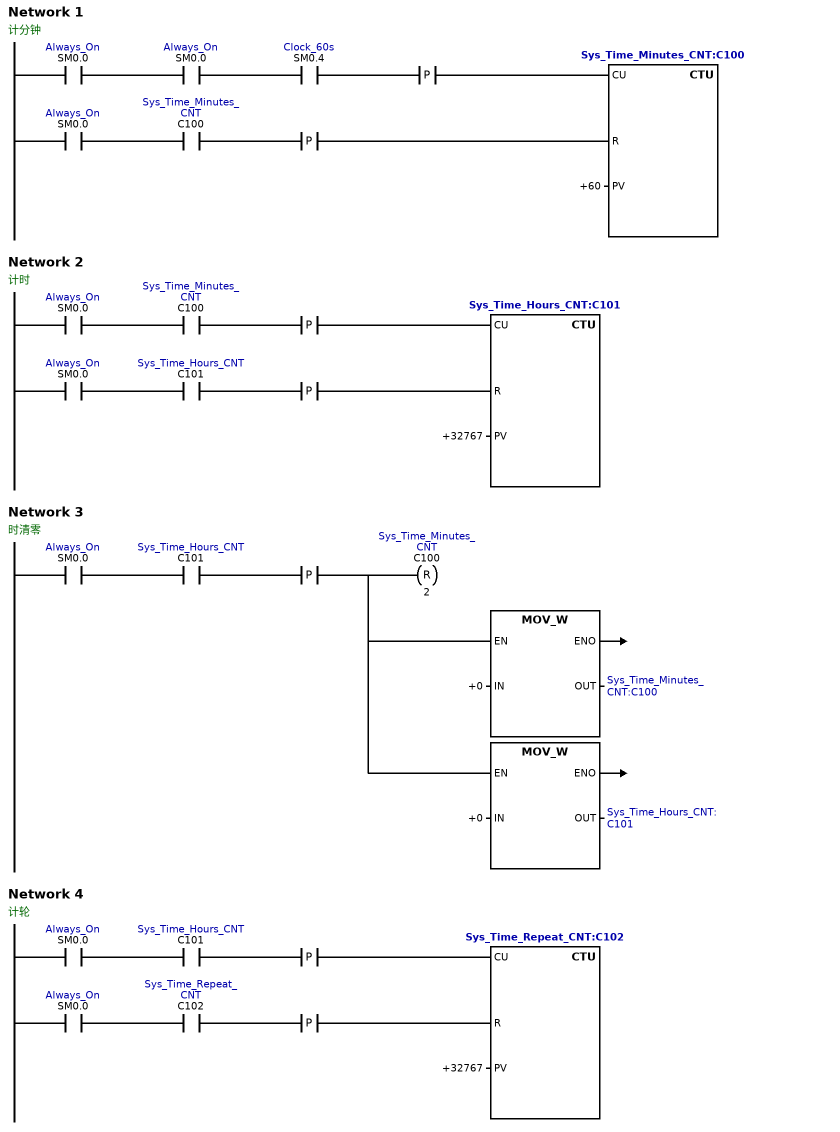
Network 1
// 计分钟
LD     Always_On:SM0.0
A      Always_On:SM0.0
A      Clock_60s:SM0.4
EU
LD     Always_On:SM0.0
A      Sys_Time_Minutes_CNT:C100
EU
CTU    Sys_Time_Minutes_CNT:C100, +60
Network 2
// 计时
LD     Always_On:SM0.0
A      Sys_Time_Minutes_CNT:C100
EU
LD     Always_On:SM0.0
A      Sys_Time_Hours_CNT:C101
EU
CTU    Sys_Time_Hours_CNT:C101, +32767
Network 3
// 时清零
LD     Always_On:SM0.0
A      Sys_Time_Hours_CNT:C101
EU
R      Sys_Time_Minutes_CNT:C100, 2
MOVW   +0, Sys_Time_Minutes_CNT:C100
MOVW   +0, Sys_Time_Hours_CNT:C101
Network 4
// 计轮
LD     Always_On:SM0.0
A      Sys_Time_Hours_CNT:C101
EU
LD     Always_On:SM0.0
A      Sys_Time_Repeat_CNT:C102
EU
CTU    Sys_Time_Repeat_CNT:C102, +32767
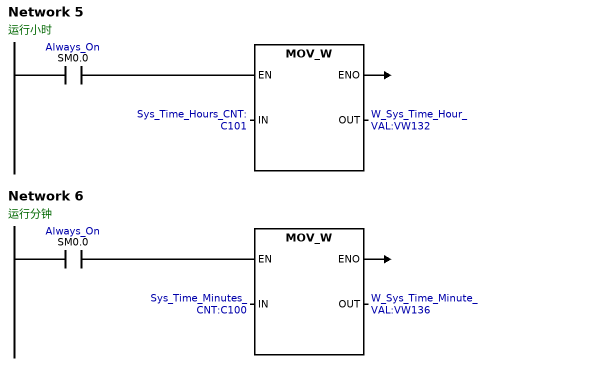
Network 5
// 运行小时
LD     Always_On:SM0.0
MOVW   Sys_Time_Hours_CNT:C101, W_Sys_Time_Hour_VAL:VW132
Network 6
// 运行分钟
LD     Always_On:SM0.0
MOVW   Sys_Time_Minutes_CNT:C100, W_Sys_Time_Minute_VAL:VW136
END_SUBROUTINE_BLOCK

SUBROUTINE_BLOCK 报警复位:SBR13
TITLE=报警复位子程序
// 功能：
// 1、报警逻辑
// 系统故障报警停机如：	
// 	检漏报警		停机
// 	空气压力低报警		停机
// 	燃气压力高报警		停机
// 	燃气压力低报警		停机
// 	点火前检测到火焰报警	停机
// 	点火失败报警		停机
// 	火焰丢失报警		停机
// 关闭所有燃气阀门：包括点火阀、主火阀、安全阀、
// 复位点火成功标志，
// 
// 调节阀故障只显示
// 	空气调节阀检测失败报警	提示
// 	燃气调节阀检测失败报警	提示
// 
// 
// 2、复位逻辑
// 复位7个故障，M20.1-M20.7
// 
// 两个调节阀故障，上电的时候才复位，这里不复位。
// 
// 
// 
BEGIN
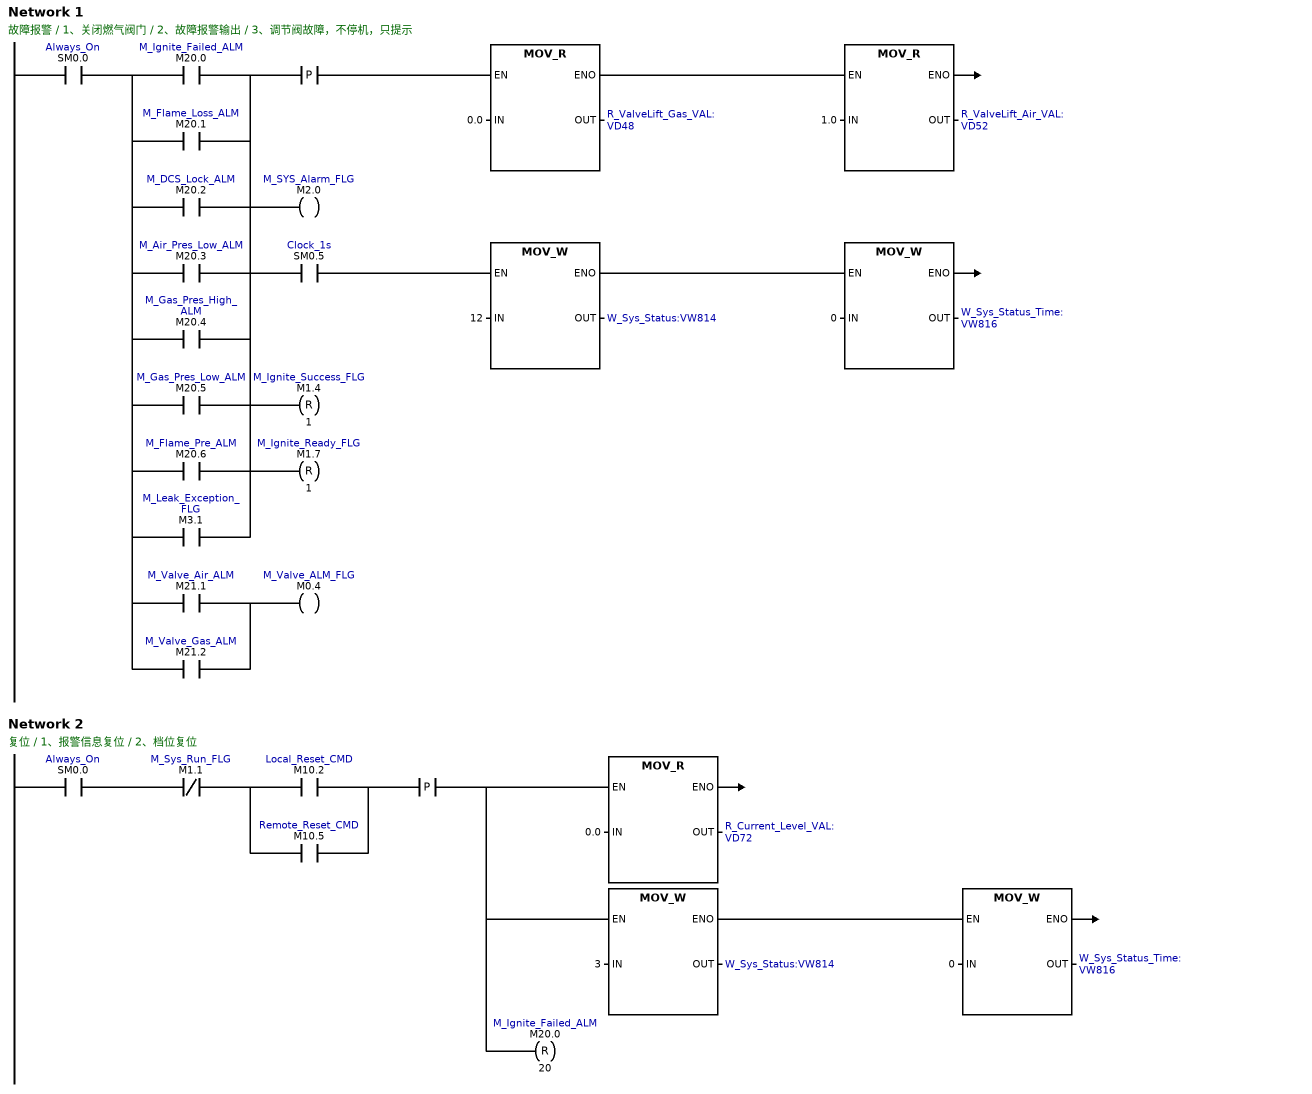
Network 1
// 故障报警
// 1、关闭燃气阀门
// 2、故障报警输出
// 3、调节阀故障，不停机，只提示
LD     Always_On:SM0.0
LPS
LD     M_Ignite_Failed_ALM:M20.0
O      M_Flame_Loss_ALM:M20.1
O      M_DCS_Lock_ALM:M20.2
O      M_Air_Pres_Low_ALM:M20.3
O      M_Gas_Pres_High_ALM:M20.4
O      M_Gas_Pres_Low_ALM:M20.5
O      M_Flame_Pre_ALM:M20.6
O      M_Leak_Exception_FLG:M3.1
ALD
LPS
EU
MOVR   0.0, R_ValveLift_Gas_VAL:VD48
AENO
MOVR   1.0, R_ValveLift_Air_VAL:VD52
LRD
=      M_SYS_Alarm_FLG:M2.0
LRD
A      Clock_1s:SM0.5
MOVW   12, W_Sys_Status:VW814
AENO
MOVW   0, W_Sys_Status_Time:VW816
LRD
R      M_Ignite_Success_FLG:M1.4, 1
LPP
R      M_Ignite_Ready_FLG:M1.7, 1
LPP
LD     M_Valve_Air_ALM:M21.1
O      M_Valve_Gas_ALM:M21.2
ALD
=      M_Valve_ALM_FLG:M0.4
Network 2
// 复位
// 1、报警信息复位
// 2、档位复位
LD     Always_On:SM0.0
AN     M_Sys_Run_FLG:M1.1
LD     Local_Reset_CMD:M10.2
O      Remote_Reset_CMD:M10.5
ALD
EU
LPS
MOVR   0.0, R_Current_Level_VAL:VD72
MOVW   3, W_Sys_Status:VW814
AENO
MOVW   0, W_Sys_Status_Time:VW816
LPP
R      M_Ignite_Failed_ALM:M20.0, 20
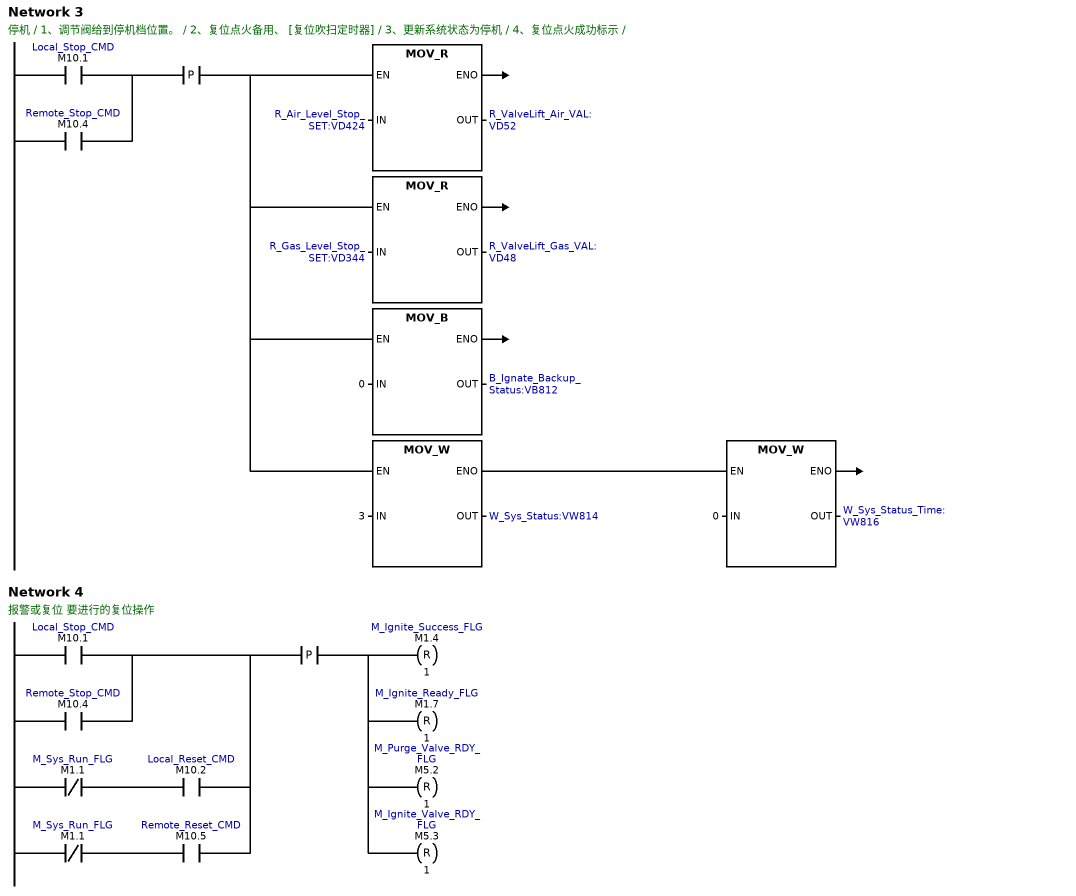
Network 3
// 停机
// 1、调节阀给到停机档位置。
// 2、复位点火备用、 [复位吹扫定时器]
// 3、更新系统状态为停机
// 4、复位点火成功标示
// 
LD     Local_Stop_CMD:M10.1
O      Remote_Stop_CMD:M10.4
EU
MOVR   R_Air_Level_Stop_SET:VD424, R_ValveLift_Air_VAL:VD52
MOVR   R_Gas_Level_Stop_SET:VD344, R_ValveLift_Gas_VAL:VD48
MOVB   0, B_Ignate_Backup_Status:VB812
MOVW   3, W_Sys_Status:VW814
AENO
MOVW   0, W_Sys_Status_Time:VW816
Network 4
// 报警或复位 要进行的复位操作
LD     Local_Stop_CMD:M10.1
O      Remote_Stop_CMD:M10.4
LDN    M_Sys_Run_FLG:M1.1
A      Local_Reset_CMD:M10.2
OLD
LDN    M_Sys_Run_FLG:M1.1
A      Remote_Reset_CMD:M10.5
OLD
EU
R      M_Ignite_Success_FLG:M1.4, 1
R      M_Ignite_Ready_FLG:M1.7, 1
R      M_Purge_Valve_RDY_FLG:M5.2, 1
R      M_Ignite_Valve_RDY_FLG:M5.3, 1
END_SUBROUTINE_BLOCK

// SBR18: protected block, not included

// SBR21: protected block, not included

// SBR22: protected block, not included

// SBR23: protected block, not included

// SBR24: protected block, not included

// SBR30: protected block, not included

// SBR31: protected block, not included

// INT0: protected block, not included

DATA_BLOCK_TAB 参数
BEGIN
         W_Purge_Time_SET, 300 //VW528, 吹扫时间设定
         W_Ignite_Delay_SET, 10 //VW532, 点火延时设定值
         W_Ignite_Spark_Time_SET, 70 //VW568, 高压包打火时长设定值
         W_Valve_Ignite_Time_SET, 10 //VW572, 点火阀开启延时设定值
         W_ValveCut_Delay_SET, 20 //VW536  主火阀(切断阀)开启延时设定值
         W_ValveDetect_Time_SET, 600 //VW576, 调节阀检测时长设定值
         R_ValveC_Step2_Per_SET, 80.0 //VD590, 调节阀检测第2步开度设定
         R_Gas_DiffAlow_SET, 5.0 //VD312, 燃气偏差允许值设定
         R_Air_DiffAlow_SET, 5.0 //VD316, 空气偏差允许值设定
         W_PreFlame_Time_SET, 20 //VW564, 前火检时长设定值
         W_Flame_Build_Time_SET, 10 //VW580, 火焰建立延时时长设定值
         W_Flame_Loss_Time_SET, 20 //VW584  火焰丢失延时时长设定值，建议1~3秒
         B_Remote_Function_SET, 0 //VB700  远程功能：0禁用远程、>1启用远程
END_DATA_BLOCK_TAB

DATA_BLOCK_TAB 空燃比
BEGIN
//数据页注释
//按 F1 获取帮助和示例数据页
         R_Stage1_Temp_SET, 0.0
         R_Stage2_Temp_SET, 0.0
         R_Stage3_Temp_SET, 0.0
         R_Stage4_Temp_SET, 0.0
         R_Stage5_Temp_SET, 0.0
         R_Stage6_Temp_SET, 500.0
         W_Stage1_Temp_Time_SET, 0
         W_Stage2_Temp_Time_SET, 0
         W_Stage3_Temp_Time_SET, 0
         W_Stage4_Temp_Time_SET, 0
         W_Stage5_Temp_Time_SET, 0
         W_Stage6_Temp_Time_SET, 1
         R_Temp_Upper_Limit_SET, 999.0
         R_Over_Temp_Stop_SET, 985.0
         R_PID_P_SET, 17.0
         R_PID_I_SET, 10.0
         R_PID_D_SET, 0
         R_PID_Ts_SET, 0.01
         R_Gas_Level1_SET, 15.0
         R_Gas_Level2_SET, 20.0
         R_Gas_Level3_SET, 30.0
         R_Gas_Level4_SET, 35.0
         R_Gas_Level5_SET, 40.0
         R_Gas_Level6_SET, 45.0
         R_Gas_Level7_SET, 50.0
         R_Gas_Level8_SET, 55.0
         R_Gas_Level9_SET, 60.0
         R_Gas_Level10_SET, 65.0
         R_Gas_Level11_SET, 70.0
         R_Gas_Level12_SET, 75.0
         R_Gas_Level13_SET, 80.0
         R_Gas_Level14_SET, 85.0
         R_Air_Level1_SET, 30.0
         R_Air_Level2_SET, 40.0
         R_Air_Level3_SET, 60.0
         R_Air_Level4_SET, 65.0
         R_Air_Level5_SET, 70.0
         R_Air_Level6_SET, 75.0
         R_Air_Level7_SET, 80.0
         R_Air_Level8_SET, 85.0
         R_Air_Level9_SET, 90.0
         R_Air_Level10_SET, 95.0
         R_Air_Level11_SET, 99.0
         R_Air_Level12_SET, 99.0
         R_Air_Level13_SET, 99.0
         R_Air_Level14_SET, 99.0
         R_Level_Total_SET, 14.0
         R_Air_Level_Ignite_SET, 10.0
         R_Purge_Valve_Air_SET, 80.0 //VD320, 吹扫空气阀开度设定值
END_DATA_BLOCK_TAB
